{attribute 'qualified_only'}
VAR_GLOBAL
	sensorPoti		AT %I*	: SensorbeckhoffIO_In;
END_VAR

(* stored: Version 1.1.0.1
   GVL IO: Id {56418916-8138-0de4-16f0-559cd50f4cfd} *)
